// TIA Portal V21 export
// export: Created 2026-07-07T08:06:08.7518199Z, ExportSetting WithReadOnly, DisplayName Totally Integrated Automation Portal, DisplayVersion V21, DisplayName SINAMICS Startdrive Advanced, DisplayVersion V21, DisplayName SINAMICS Startdrive G110M, G120, G120C, G120D, G120P, G115D, DisplayVersion V21, DisplayName SINAMICS Startdrive G130, G150, S120, S150, G200, G220, S200, S210, S220, Innomotics MVD, DisplayVersion V21, DisplayName STEP 7 Professional, DisplayVersion V21, DisplayName STEP 7 Safety, DisplayVersion V21, DisplayName Tech WebApplication, DisplayVersion V21, DisplayName WinCC Basic/Comfort/Advanced, DisplayVersion V21, DisplayName WinCC Professional, DisplayVersion V21, DisplayName WinCC Unified, DisplayVersion V21
FUNCTION "FC_ModeInterlock_LAD" : Void   // FC2, LAD
{ S7_Optimized_Access := 'TRUE' }
// stored: CodeModifiedDate 2026-07-07T08:05:43.3025456Z, CompileDate 2026-07-07T08:05:44.4848578Z, CreationDate 2026-07-07T08:05:43.2800733Z, DownloadDate 0001-01-01T00:00:00Z, InterfaceModifiedDate 2026-07-07T08:05:43.2800733Z, IsConsistent true, LibraryConformanceStatus 警告： 该对象包含对全局数据块的访问。, LoadMemoryLength 5413, ModifiedDate 2026-07-07T08:05:43.3386166Z, PLCSimAdvancedSupport true, ParameterModified 2026-07-07T08:05:43.2800733Z, SetENOAutomatically false, StructureModified 2026-07-07T08:05:43.2800733Z, WorkMemoryLength 76
BEGIN

REGION Network 1: Manual active interlock
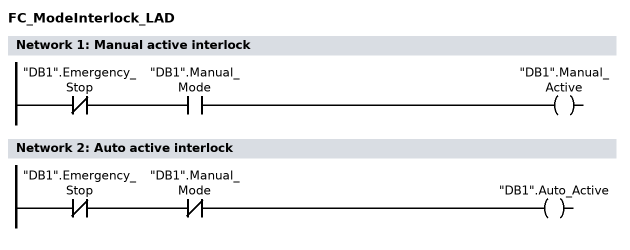
   RUNG wire#powerrail
      I_Contact( "DB1".Emergency_Stop )
      Contact( "DB1".Manual_Mode )
      Coil( "DB1".Manual_Active )
   END_RUNG
   // the same network as SCL:
   "DB1".Manual_Active := NOT "DB1".Emergency_Stop AND "DB1".Manual_Mode;
END_REGION

REGION Network 2: Auto active interlock
   RUNG wire#powerrail
      I_Contact( "DB1".Emergency_Stop )
      I_Contact( "DB1".Manual_Mode )
      Coil( "DB1".Auto_Active )
   END_RUNG
   // the same network as SCL:
   "DB1".Auto_Active := NOT "DB1".Emergency_Stop AND NOT "DB1".Manual_Mode;
END_REGION
END_FUNCTION
